Staubli VAL3: realTimeCtrl.pjx

--- realTimeCtrl.pjx ---
Parameters version=s7.9.1 stackSize=500000 millimeterUnit=true
Program file=ASCIItoNum.pgx
Program file=calcForce.pgx
Program file=dataFileOutput.pgx
Program file=dataUpdate.pgx
Program file=initSensor.pgx
Program file=loopReadForce.pgx
Program file=modelParmIdent.pgx
Program file=newCommand.pgx
Program file=readDeteVal.pgx
Program file=robotMove.pgx
Program file=robotPlanner.pgx
Program file=robotStateInq.pgx
Program file=start.pgx
Program file=stop.pgx
Program file=userInterface.pgx
Data file=realTimeCtrl.dtx

--- start.pgx ---
program start()
  local jointRx l_jInitPoint
  local jointRx l_jStartPoint
  local num l_nNum
  local string l_sConnect
begin

  //===================== 程序说明 =====================
  //Goal: 改程序用于Staubli TX90机器人的实时导纳控制，即通过外部传感器输入的力信息，经过阻抗模型转换成控制机器人的位置指令，
  //用来控制机器人的运动。本程序要实现的目标是，通过拖拽机器人到目标位置。
  //Author: Jade Cong
  //Date: 2017-05-26

  //Modification:
  //Modification Time:



  //===================== 第一步：初始化设备（机器人，传感器），并确保无任何问题 =====================
  //---------- 清理用户界面（清楚上一次程序终止后残留的用户界面信息） -----------
  cls()


  //----------- 初始化机器人（移动机器人至初始位置，并进入Sychronous Movej模式） ----------
  //移动机器人至初始零位置（从上一次程序结束后的位置恢复，防止干扰下一次程序执行）
  l_jInitPoint={0,0,0,0,0,0}
  resetMotion(l_jInitPoint)
  autoConnectMove(bActive)

  //移动机器人至运动开始准备点（准备从当前位置进入同步模式）
  l_jStartPoint={50,40,75,0,65,0}
  movej(l_jStartPoint,flange,mMdesc_Init)
  waitEndMove()

  //开始Sychronous Movej运动模式，并检测是否成功（注意运动参数mMdesc_RT的设置，其控制机器人的最大速度和加速度）
  $movejSyncBegin(mMdesc_RT)

  //等待机器人接近Sychronous Movej实时运动模式的开始点（为避免机器人运动突然大距离运动而报错，故此点不能离当前点太远）
  jJoint_RT_Start={50.01,40,75,0,65,0}
  wait($movejSync(jJoint_RT_Start)==true)

  //返回Sychronous Movej当前的运动状态
  if $movejSyncState()==1
    popUpMsg("MovejSynch running, no error!")
  elseIf $movejSyncState()==0
    popUpMsg("MovejSynch not started!")
    wait($movejSync(jJoint_RT_Start)==true)
  elseIf $movejSyncState()==2
    popUpMsg("MovejSynch stopped in error(after invalid command)!")
    $movejSyncEnd()
  elseIf $movejSyncState()==3
    popUpMsg("MovejSynch runing, last command was not refreshed in time!")
    $movejSyncEnd()
  elseIf $movejSyncState()==4
    popUpMsg("MovejSynch runing, commands are locked because motion is stopped!")
    $movejSyncEnd()
  endIf


  //----------- 初始化传感器（完成通讯及零点校准），并检测是否成功 -----------
  call initSensor("io:Wacoh",l_sConnect)
  if l_sConnect=="yes"
    putln("Connection success!")
    delay(1.0)
  else
    putln("Connection fail!")
    delay(1.0)
  endIf



  //===================== 第二步：周期性更新位置指令并送给机器人执行，同时采集、更新并输出、输入数据（4ms） ====================
  //---------- 确定机器人及传感器的初始状态（当前和期望）和模型（阻抗/other）参数，用于第一次更新机器人位置指令 ----------
  //阻抗参数
  for l_nNum=0 to 2
    nMass[l_nNum,l_nNum]=0.1
    nDamp[l_nNum,l_nNum]=4
    nStiffness[l_nNum,l_nNum]=4

    nMass[l_nNum+3,l_nNum+3]=0.00001
    nDamp[l_nNum+3,l_nNum+3]=4
    nStiffness[l_nNum+3,l_nNum+3]=4
  endFor

  //当前状态
  nForceTorque=0
  pNowPointPos=$getPosFbk(flange,world)
  nNowPointVel=0
  nNowPointAccel=0

  //期望状态
  ndForceTorque=0
  pdPointPos=pNowPointPos
  ndPointVel=0
  ndPointAccel=0


  //---------- 创建同步任务，每4ms更新机器人的位置指令（根据上一次采集的数据对下一次的运动产生修正） ----------
  taskCreateSync "newCommand",0.004,bOverRun[0],newCommand(pPointCommand)


  //---------- 创建同步任务，每4ms机器人执行新的位置指令 ----------
  taskCreateSync "robotMove",0.004,bOverRun[1],robotMove(pPointCommand)


  //---------- 创建同步任务，每4ms实时进行数据采集、更新，并输出（传感器及机器人状态）;输入并更新（阻抗模型参数，机器人运动规划所期望的Force/Motion State） ----------
  //首先创建文件，其次循环写入（输出）、读取（输入）数据
  //  nFileID[0]=$fileOpen("Disk://Cache Data/Sensor_Data.txt","w")
  //  nFileID[1]=$fileOpen("Disk://Cache Data/Robot_Cartesian_Data.txt","w")
  //  nFileID[2]=$fileOpen("Disk://Cache Data/Robot_Joint_Data.txt","w")

  //nFileID[3]=$fileOpen("Disk:///Cache Data/Desired_Sensor_Data.txt","r")
  //nFileID[4]=$fileOpen("Disk://Cache Data/Desired_Robot_Cartesian_Data.txt","r")
  //nFileID[5]=$fileOpen("Disk://Cache Data/Desired_Robot_Joint_Data.txt","r")

  //  if nFileID[0]>=0 and nFileID[1]>=0 and nFileID[2]>=0
  //    popUpMsg("Files open success!")
  //  else
  //    popUpMsg("Files open fail!")
  //  endIf

  //更新（输入，输出）数据
  taskCreateSync "dataUpdate",0.004,bOverRun[2],dataUpdate(nFileID)



  //==================== 第三步：实时更新显示并监测机器人及传感器的状态 ====================
  //创建异步任务，显示更新传感数据（力/力矩）和机器人当前状态（位置，速度，加速度）
  taskCreate "userInterface",20,userInterface(nForceTorque,pNowPointPos,nNowPointVel,nNowPointAccel,jNowJointPos,nNowJointVel,nNowJointAccel)

end

--- dataFileOutput.pgx ---
public program dataFileOutput(num& x_nFileID[], num& x_nForceTorque[], pointRx& x_pNowPointPos[], num& x_nNowPointVel[], num& x_nNowPointAcce[], jointRx& x_jNowJointPos[], num& x_nNowJointVel[], num& x_nNowJointAcce[])
  local num l_nNowJointPos[6]
  local num l_nNowPointPos[6]
begin

  //==================== 输出需要的数据（机器人、传感器的状态）到文件，用于机器人模型参数辨识、分析及规划控制 ====================

  //写入传感器数据到文件1
  $fileSet(x_nFileID[0],x_nForceTorque[0],6)

  //写入机器人笛卡尔空间下（Cartesian Space）数据到文件2
  l_nNowPointPos[0]=x_pNowPointPos.trsf.x
  l_nNowPointPos[1]=x_pNowPointPos.trsf.y
  l_nNowPointPos[2]=x_pNowPointPos.trsf.z
  l_nNowPointPos[3]=x_pNowPointPos.trsf.rx
  l_nNowPointPos[4]=x_pNowPointPos.trsf.ry
  l_nNowPointPos[5]=x_pNowPointPos.trsf.rz

  $fileSet(x_nFileID[1],l_nNowPointPos[0],6)
  $fileSet(x_nFileID[1],x_nNowPointVel[0],6)
  $fileSet(x_nFileID[1],x_nNowPointAcce[0],6)

  //写入机器人关节空间下（Joint Space）数据到文件3
  l_nNowJointPos[0]=x_jNowJointPos.j1
  l_nNowJointPos[1]=x_jNowJointPos.j2
  l_nNowJointPos[2]=x_jNowJointPos.j3
  l_nNowJointPos[3]=x_jNowJointPos.j4
  l_nNowJointPos[4]=x_jNowJointPos.j5
  l_nNowJointPos[5]=x_jNowJointPos.j6

  $fileSet(x_nFileID[2],l_nNowJointPos[0],6)
  $fileSet(x_nFileID[2],x_nNowJointVel[0],6)
  $fileSet(x_nFileID[2],x_nNowJointAcce[0],6)

end

--- modelParmIdent.pgx ---
public program modelParmIdent(num& x_nMass[] (dimensions=2), num& x_nDamp[] (dimensions=2), num& x_nStiffness[] (dimensions=2))
begin

  //==================== 实时在线辨识机器人（阻抗/other）模型参数（待补充），当前使用假定辨识参数 ====================

  //---------- 阻抗模型参数在线辨识（待补充） ----------



  //---------- 当前假定阻抗模型参数（位置+姿态）（注意单位换算，当前使用MKS） ----------
  //质量参数M（N*s^2/m,N*s^2/°）
  x_nMass[0,0]=0.1
  x_nMass[1,1]=0.1
  x_nMass[2,2]=0.1

  x_nMass[3,3]=0.00005
  x_nMass[4,4]=0.00005
  x_nMass[5,5]=0.00005

  //阻尼参数B（N*s/m,N*s/°）
  x_nDamp[0,0]=4
  x_nDamp[1,1]=4
  x_nDamp[2,2]=4

  x_nDamp[3,3]=4
  x_nDamp[4,4]=4
  x_nDamp[5,5]=4

  //刚度参数K（N/m,N/°）
  x_nStiffness[0,0]=4
  x_nStiffness[1,1]=4
  x_nStiffness[2,2]=4

  x_nStiffness[3,3]=4
  x_nStiffness[4,4]=4
  x_nStiffness[5,5]=4

end

--- userInterface.pgx ---
public program userInterface(num& x_nFTData[], pointRx& x_pPointPos[], num& x_nPointVel[], num& x_nPointAccel[], jointRx& x_jJointPos[], num& x_nJointVel[], num& x_nJointAccel[])
begin

  //===================== 更新显示传感器数据和机器人当前状态 =====================

  //启动用户界面
  userPage()


  //循环显示数据
  while true

    //清理用户界面
    cls()


    //显示传感器数据
    //gotoxy(0,7)
    putln("Force/Torque Sensor Data")

    //gotoxy(1,0)
    put("Fx:")
    putln(x_nFTData[0])
    //gotoxy(1,13)
    put("Fy:")
    putln(x_nFTData[1])
    //gotoxy(1,26)
    put("Fz:")
    putln(x_nFTData[2])

    //gotoxy(2,0)
    put("Mx:")
    putln(x_nFTData[3])
    //gotoxy(2,13)
    put("My:")
    putln(x_nFTData[4])
    //gotoxy(2,26)
    put("Mz:")
    putln(x_nFTData[5])


    //显示机器人状态（位置，速度，加速度/关节位置，速度，加速度）
    //gotoxy(4,9)
    putln("Robot Current State")

    //Cartesian Position
    //gotoxy(5,0)
    put("X:")
    putln(x_pPointPos.trsf.x)
    //gotoxy(5,13)
    put("Y:")
    putln(x_pPointPos.trsf.y)
    //gotoxy(5,26)
    put("Z:")
    putln(x_pPointPos.trsf.z)

    //gotoxy(6,0)
    put("Rx:")
    putln(x_pPointPos.trsf.rx)
    //gotoxy(6,13)
    put("Ry:")
    putln(x_pPointPos.trsf.ry)
    //gotoxy(6,26)
    put("Rz:")
    putln(x_pPointPos.trsf.rz)


//    //显示传感器数据
//    gotoxy(0,7)
//    putln("Force/Torque Sensor Data")
//
//    gotoxy(1,0)
//    put("Fx:")
//    put(x_nFTData[0])
//    gotoxy(1,13)
//    put("Fy:")
//    put(x_nFTData[1])
//    gotoxy(1,26)
//    put("Fz:")
//    put(x_nFTData[2])
//
//    gotoxy(2,0)
//    put("Mx:")
//    put(x_nFTData[3])
//    gotoxy(2,13)
//    put("My:")
//    put(x_nFTData[4])
//    gotoxy(2,26)
//    put("Mz:")
//    put(x_nFTData[5])
//
//
//    //显示机器人状态（位置，速度，加速度/关节位置，速度，加速度）
//    gotoxy(4,9)
//    putln("Robot Current State")
//
//    //Cartesian Position
//    gotoxy(5,0)
//    put("X:")
//    put(x_pPointPos.trsf.x)
//    gotoxy(5,13)
//    put("Y:")
//    put(x_pPointPos.trsf.y)
//    gotoxy(5,26)
//    put("Z:")
//    put(x_pPointPos.trsf.z)
//
//    gotoxy(6,0)
//    put("Rx:")
//    put(x_pPointPos.trsf.rx)
//    gotoxy(6,13)
//    put("Ry:")
//    put(x_pPointPos.trsf.ry)
//    gotoxy(6,26)
//    put("Rz:")
//    put(x_pPointPos.trsf.rz)
//
//    //Cartesian Velocity
//    gotoxy(7,0)
//    put("X':")
//    put(x_nPointVel[0])
//    gotoxy(7,13)
//    put("Y':")
//    put(x_nPointVel[1])
//    gotoxy(7,26)
//    put("Z':")
//    put(x_nPointVel[2])
//
//    gotoxy(8,0)
//    put("Rx':")
//    put(x_nPointVel[3])
//    gotoxy(8,13)
//    put("Ry':")
//    put(x_nPointVel[4])
//    gotoxy(8,26)
//    put("Rz':")
//    put(x_nPointVel[5])
//
//    //Joint Position
//    gotoxy(9,0)
//    put("J1:")
//    put(x_jJointPos.j1)
//    gotoxy(9,13)
//    put("J2:")
//    put(x_jJointPos.j2)
//    gotoxy(9,26)
//    put("J3:")
//    put(x_jJointPos.j3)
//
//    gotoxy(10,0)
//    put("J4:")
//    putln(x_jJointPos.j4)
//    gotoxy(10,13)
//    put("J5:")
//    putln(x_jJointPos.j5)
//    gotoxy(10,26)
//    put("J6:")
//    putln(x_jJointPos.j6)
//
//    //Joint Velocity
//    gotoxy(11,0)
//    put("J1':")
//    put(x_nJointVel[0])
//    gotoxy(11,13)
//    put("J2':")
//    put(x_nJointVel[1])
//    gotoxy(11,26)
//    put("J3':")
//    put(x_nJointVel[2])
//
//    gotoxy(12,0)
//    put("J4':")
//    put(x_nJointVel[3])
//    gotoxy(12,13)
//    put("J5':")
//    put(x_nJointVel[4])
//    gotoxy(12,26)
//    put("J6':")
//    put(x_nJointVel[5])


    //强制结束当前任务，进入下一次sequence循环
    delay(0.0)

  endWhile

end
